(* Schneider Machine Expert - Basic project INTEGRATED_3_CONVEYOR_TM221CE24R_REV3, file version 3.0.0.0 *)
(* ProjectInformations: Name=New project *)

HARDWARE
  Cpu 0: TM221CE24R
  ModuleExtensionObject 0: TM3DI32K
  ModuleExtensionObject 1: TM3AI2H/G
  EthernetConfiguration: NetworkName=M221, IpAllocationMode=FixedAddress, IpAddress=0.0.0.0, SubnetMask=0.0.0.0
  SerialLineConfiguration: Baud=Baud19200, Parity=ParityEven, DataBits=DataBits8, StopBits=StopBits1, PhysicalMedium=PhysicalMediumRs485, TransmissionMode=TransmissionModeModbusRtu, SlaveId=1, Addressing=SlaveAddressing
  MastTask: UsePeriodScanMode=false, PeriodScan=100
  FastTask: Period=255
  CpuBehavior: StartingMode=StartAsPreviousState, AutoSaveRamOnEeprom=true, WatchdogPeriod=250

SYMBOLS  (address, symbol, comment, settings)
  %M0       AUTO_MODE  "1 Auto"
  %M1       START_HMI  "Start HMI"
  %M2       STOP_HMI  "Stop HMI"
  %M3       JOG_INFEED  "Jog infeed"
  %M4       JOG_TRANSFER  "Jog transfer"
  %M5       JOG_OUTFEED  "Jog outfeed"
  %M6       RESET_HMI  "Reset HMI"
  %M7       MAINTENANCE_ENABLE  "Izin maintenance"
  %M10      SYSTEM_RUN  "Latch produksi"
  %M11      SAFETY_OK  "Ringkasan interlock"
  %M12      OUTFEED_AUTO_CMD  "Auto command outfeed"
  %M13      TRANSFER_AUTO_CMD  "Auto command transfer"
  %M14      INFEED_AUTO_CMD  "Auto command infeed"
  %M15      INFEED_FINAL_CMD  "Final infeed"
  %M16      TRANSFER_FINAL_CMD  "Final transfer"
  %M17      OUTFEED_FINAL_CMD  "Final outfeed"
  %M20      TRANSFER_STAGE_READY  "Start delay transfer selesai"
  %M21      INFEED_STAGE_READY  "Start delay infeed selesai"
  %M22      REJECT_REQUEST  "Permintaan reject"
  %M23      REJECT_ACTIVE  "Solenoid reject aktif"
  %M24      PRODUCT_REJECTED  "Produk saat ini reject"
  %M25      EXIT_PULSE  "Pulsa exit"
  %M26      RESET_REQUEST  "Gabungan reset"
  %M30      JAM_INFEED  "Jam infeed"
  %M31      JAM_TRANSFER  "Jam transfer"
  %M32      JAM_OUTFEED  "Jam outfeed"
  %M33      REJECT_NOT_HOME  "Pusher gagal home"
  %M34      ALARM_ACTIVE  "Alarm umum"
  %M40      RESET_COUNTERS_HMI  "Reset counter produksi"
  %M41      MANUAL_INFEED_CMD  "Jog infeed tervalidasi"
  %M42      MANUAL_TRANSFER_CMD  "Jog transfer tervalidasi"
  %M43      MANUAL_OUTFEED_CMD  "Jog outfeed tervalidasi"
  %S5       SB_TB100MS  "Time base of 100 ms generated by an internal clock"
  %S6       SB_TB1S  "Time base of 1 s generated by an internal clock"
  %S13      SB_FIRSTRUN  "Indicates the first controller cycle in RUN mode"
  %MW1      WATER_RANGE_MM  "Range sensor level mm"
  %MW2      LEVEL_RAW_COPY  "Salinan raw input level"
  %MW10     MAX_HEIGHT_G1_MM  "Tinggi maksimum pintu 1 mm"
  %MW11     MAX_HEIGHT_G2_MM  "Tinggi maksimum pintu 2 mm"
  %MW12     MAX_HEIGHT_G3_MM  "Tinggi maksimum pintu 3 mm"
  %MW13     DEADBAND_PCT  "Deadband posisi persen"
  %MW20     ENC_ZERO_G1  "Nilai encoder pintu 1 saat tertutup"
  %MW21     ENC_ZERO_G2  "Nilai encoder pintu 2 saat tertutup"
  %MW22     ENC_ZERO_G3  "Nilai encoder pintu 3 saat tertutup"
  %MW23     ENC_SPAN_G1  "Span count tertutup-terbuka G1"
  %MW24     ENC_SPAN_G2  "Span count tertutup-terbuka G2"
  %MW25     ENC_SPAN_G3  "Span count tertutup-terbuka G3"
  %MW30     ENC_BINARY_G1  "Nilai biner encoder G1"
  %MW31     ENC_BINARY_G2  "Nilai biner encoder G2"
  %MW32     ENC_BINARY_G3  "Nilai biner encoder G3"
  %MW33     POS_COUNT_G1  "Count posisi terkoreksi G1"
  %MW34     POS_COUNT_G2  "Count posisi terkoreksi G2"
  %MW35     POS_COUNT_G3  "Count posisi terkoreksi G3"
  %MW50     TARGET_PCT_G1  "Target bukaan G1 0-100 persen"
  %MW51     TARGET_PCT_G2  "Target bukaan G2 0-100 persen"
  %MW52     TARGET_PCT_G3  "Target bukaan G3 0-100 persen"
  %MF60     POSITION_G1_PCT  "Posisi G1 persen"
  %MF62     POSITION_G2_PCT  "Posisi G2 persen"
  %MF64     POSITION_G3_PCT  "Posisi G3 persen"
  %MF66     POSITION_G1_MM  "Posisi G1 mm"
  %MF68     POSITION_G2_MM  "Posisi G2 mm"
  %MF70     POSITION_G3_MM  "Posisi G3 mm"
  %MF72     WATER_LEVEL_MM  "Level air mm"
  %MF74     WATER_LEVEL_PCT  "Level air persen"
  %MF76     WATER_RANGE_REAL  "Range level dalam REAL"
  %MF80     TARGET_G1_REAL  "Target G1 dalam REAL"
  %MF82     TARGET_G2_REAL  "Target G2 dalam REAL"
  %MF84     TARGET_G3_REAL  "Target G3 dalam REAL"
  %MF86     DEADBAND_REAL  "Deadband dalam REAL"
  %MF88     OPEN_THRESHOLD_G1  "Ambang buka G1"
  %MF90     CLOSE_THRESHOLD_G1  "Ambang tutup G1"
  %MF92     OPEN_THRESHOLD_G2  "Ambang buka G2"
  %MF94     CLOSE_THRESHOLD_G2  "Ambang tutup G2"
  %MF96     OPEN_THRESHOLD_G3  "Ambang buka G3"
  %MF98     CLOSE_THRESHOLD_G3  "Ambang tutup G3"
  %C0       TRANSFER_START_TICKS  "10 x 100 ms = 1 s"
  %C1       INFEED_START_TICKS  "10 x 100 ms = 1 s"
  %C2       REJECT_POSITION_TICKS  "5 x 100 ms = 0.5 s"
  %C3       REJECT_PULSE_TICKS  "7 x 100 ms = 0.7 s"
  %C4       JAM_INFEED_SECONDS  "10 x 1 s"
  %C5       JAM_TRANSFER_SECONDS  "10 x 1 s"
  %C6       JAM_OUTFEED_SECONDS  "10 x 1 s"
  %C7       REJECT_HOME_SECONDS  "3 x 1 s"
  %C8       GOOD_PRODUCT_COUNT  "Counter produk OK"
  %C9       REJECT_PRODUCT_COUNT  "Counter produk reject"
  %I0.0     START_PB  "Tombol Start NO"
  %I0.1     STOP_OK  "Kontak Stop NC; 1 sehat"
  %I0.2     ESTOP_OK  "Feedback safety relay; 1 sehat"
  %I0.3     OL_INFEED_OK  "Overload infeed; 1 sehat"
  %I0.4     OL_TRANSFER_OK  "Overload transfer; 1 sehat"
  %I0.5     OL_OUTFEED_OK  "Overload outfeed; 1 sehat"
  %I0.6     SENSOR_INFEED  "Sensor infeed"
  %I0.7     SENSOR_BUFFER1  "Sensor buffer 1"
  %I0.8     SENSOR_BUFFER2  "Sensor buffer 2"
  %I0.9     SENSOR_INSPECTION  "Sensor inspeksi"
  %I0.10    QUALITY_OK  "Hasil inspeksi OK"
  %I0.11    REJECT_HOME  "Pusher reject home"
  %I0.12    EXIT_SENSOR  "Sensor keluar"
  %I0.13    RESET_PB  "Reset alarm"
  %Q0.0     MOTOR_INFEED  "Motor conveyor infeed"
  %Q0.1     MOTOR_TRANSFER  "Motor conveyor transfer"
  %Q0.2     MOTOR_OUTFEED  "Motor conveyor outfeed"
  %Q0.3     REJECT_SOLENOID  "Solenoid reject"
  %Q0.4     BUZZER  "Buzzer fault"
  %Q0.5     LAMP_RUN  "Lampu run"
  %Q0.6     LAMP_MAINTENANCE  "Lampu maintenance"
  %Q0.7     LAMP_FAULT  "Lampu fault"
  %Q0.8       "Tidak digunakan"
  %Q0.9       "Tidak digunakan"
  %I1.0     ENC_G1_GRAY_B0  "E6CP pintu 1 Gray bit 0"
  %I1.1     ENC_G1_GRAY_B1  "E6CP pintu 1 Gray bit 1"
  %I1.2     ENC_G1_GRAY_B2  "E6CP pintu 1 Gray bit 2"
  %I1.3     ENC_G1_GRAY_B3  "E6CP pintu 1 Gray bit 3"
  %I1.4     ENC_G1_GRAY_B4  "E6CP pintu 1 Gray bit 4"
  %I1.5     ENC_G1_GRAY_B5  "E6CP pintu 1 Gray bit 5"
  %I1.6     ENC_G1_GRAY_B6  "E6CP pintu 1 Gray bit 6"
  %I1.7     ENC_G1_GRAY_B7  "E6CP pintu 1 Gray bit 7"
  %I1.8     ENC_G2_GRAY_B0  "E6CP pintu 2 Gray bit 0"
  %I1.9     ENC_G2_GRAY_B1  "E6CP pintu 2 Gray bit 1"
  %I1.10    ENC_G2_GRAY_B2  "E6CP pintu 2 Gray bit 2"
  %I1.11    ENC_G2_GRAY_B3  "E6CP pintu 2 Gray bit 3"
  %I1.12    ENC_G2_GRAY_B4  "E6CP pintu 2 Gray bit 4"
  %I1.13    ENC_G2_GRAY_B5  "E6CP pintu 2 Gray bit 5"
  %I1.14    ENC_G2_GRAY_B6  "E6CP pintu 2 Gray bit 6"
  %I1.15    ENC_G2_GRAY_B7  "E6CP pintu 2 Gray bit 7"
  %I1.16    ENC_G3_GRAY_B0  "E6CP pintu 3 Gray bit 0"
  %I1.17    ENC_G3_GRAY_B1  "E6CP pintu 3 Gray bit 1"
  %I1.18    ENC_G3_GRAY_B2  "E6CP pintu 3 Gray bit 2"
  %I1.19    ENC_G3_GRAY_B3  "E6CP pintu 3 Gray bit 3"
  %I1.20    ENC_G3_GRAY_B4  "E6CP pintu 3 Gray bit 4"
  %I1.21    ENC_G3_GRAY_B5  "E6CP pintu 3 Gray bit 5"
  %I1.22    ENC_G3_GRAY_B6  "E6CP pintu 3 Gray bit 6"
  %I1.23    ENC_G3_GRAY_B7  "E6CP pintu 3 Gray bit 7"
  %I1.24    MODE_AUTO  "Selector 1=AUTO 0=MANUAL"
  %I1.25    MAN_OPEN_G1  "PB manual buka pintu 1"
  %I1.26    MAN_CLOSE_G1  "PB manual tutup pintu 1"
  %I1.27    MAN_OPEN_G2  "PB manual buka pintu 2"
  %I1.28    MAN_CLOSE_G2  "PB manual tutup pintu 2"
  %I1.29    MAN_OPEN_G3  "PB manual buka pintu 3"
  %I1.30    MAN_CLOSE_G3  "PB manual tutup pintu 3"
  %I1.31    RESET_FAULT  "PB reset fault"
  %IW2.0    LEVEL_RAW  "Sensor level 4-20 mA raw 4000-20000"  [Type=Type_4_20mA, Scope=Scope_Customized, Minimum=4000, Maximum=20000]

POU INTEGRATED_3_CONVEYOR_IL
  (* SectionNumber=1 *)

// Rung 0: N01_SAFETY
// Stop, E-Stop, dan tiga overload.
  LD %I0.1                (* STOP_OK *)
  AND %I0.2               (* ESTOP_OK *)
  AND %I0.3               (* OL_INFEED_OK *)
  AND %I0.4               (* OL_TRANSFER_OK *)
  AND %I0.5               (* OL_OUTFEED_OK *)
  ANDN %M2                (* STOP_HMI *)
  ST %M11                 (* SAFETY_OK *)
  // as ST:
  //   SAFETY_OK := STOP_OK AND ESTOP_OK AND OL_INFEED_OK AND OL_TRANSFER_OK AND OL_OUTFEED_OK AND NOT STOP_HMI;

// Rung 1: N02_SYSTEM_RUN
// Latch produksi Auto.
  LD %I0.0                (* START_PB *)
  OR %M1                  (* START_HMI *)
  OR %M10                 (* SYSTEM_RUN *)
  AND %M0                 (* AUTO_MODE *)
  AND %M11                (* SAFETY_OK *)
  ST %M10                 (* SYSTEM_RUN *)
  // as ST:
  //   SYSTEM_RUN := (START_PB OR START_HMI OR SYSTEM_RUN) AND AUTO_MODE AND SAFETY_OK;

// Rung 2: N03_RESET
// Gabungan reset.
  LD %I0.13               (* RESET_PB *)
  OR %M6                  (* RESET_HMI *)
  ST %M26                 (* RESET_REQUEST *)
  // as ST:
  //   RESET_REQUEST := RESET_PB OR RESET_HMI;

// Rung 3: N04_OUTFEED_BASE
// Hilir start lebih dahulu.
  LD %M10                 (* SYSTEM_RUN *)
  ANDN %M34               (* ALARM_ACTIVE *)
  ST %M12                 (* OUTFEED_AUTO_CMD *)
  // as ST:
  //   OUTFEED_AUTO_CMD := SYSTEM_RUN AND NOT ALARM_ACTIVE;

// Rung 4: N05_PRESET_C0
// Preset transfer start.
  LD %S13                 (* SB_FIRSTRUN *)
  [ %C0.P := 10 ]         (* TRANSFER_START_TICKS *)
  // as ST:
  //   IF SB_FIRSTRUN THEN TRANSFER_START_TICKS.P := 10; END_IF;

// Rung 5: N05_PRESET_C1
// Preset infeed start.
  LD %S13                 (* SB_FIRSTRUN *)
  [ %C1.P := 10 ]         (* INFEED_START_TICKS *)
  // as ST:
  //   IF SB_FIRSTRUN THEN INFEED_START_TICKS.P := 10; END_IF;

// Rung 6: N05_PRESET_C2
// Preset posisi reject.
  LD %S13                 (* SB_FIRSTRUN *)
  [ %C2.P := 5 ]          (* REJECT_POSITION_TICKS *)
  // as ST:
  //   IF SB_FIRSTRUN THEN REJECT_POSITION_TICKS.P := 5; END_IF;

// Rung 7: N05_PRESET_C3
// Preset pulsa reject.
  LD %S13                 (* SB_FIRSTRUN *)
  [ %C3.P := 7 ]          (* REJECT_PULSE_TICKS *)
  // as ST:
  //   IF SB_FIRSTRUN THEN REJECT_PULSE_TICKS.P := 7; END_IF;

// Rung 8: N05_PRESET_C4
// Preset jam infeed.
  LD %S13                 (* SB_FIRSTRUN *)
  [ %C4.P := 10 ]         (* JAM_INFEED_SECONDS *)
  // as ST:
  //   IF SB_FIRSTRUN THEN JAM_INFEED_SECONDS.P := 10; END_IF;

// Rung 9: N05_PRESET_C5
// Preset jam transfer.
  LD %S13                 (* SB_FIRSTRUN *)
  [ %C5.P := 10 ]         (* JAM_TRANSFER_SECONDS *)
  // as ST:
  //   IF SB_FIRSTRUN THEN JAM_TRANSFER_SECONDS.P := 10; END_IF;

// Rung 10: N05_PRESET_C6
// Preset jam outfeed.
  LD %S13                 (* SB_FIRSTRUN *)
  [ %C6.P := 10 ]         (* JAM_OUTFEED_SECONDS *)
  // as ST:
  //   IF SB_FIRSTRUN THEN JAM_OUTFEED_SECONDS.P := 10; END_IF;

// Rung 11: N05_PRESET_C7
// Preset pusher home.
  LD %S13                 (* SB_FIRSTRUN *)
  [ %C7.P := 3 ]          (* REJECT_HOME_SECONDS *)
  // as ST:
  //   IF SB_FIRSTRUN THEN REJECT_HOME_SECONDS.P := 3; END_IF;

// Rung 12: N06_TRANSFER_DELAY
// Delay 1 detik.
  BLK %C0                 (* TRANSFER_START_TICKS *)
  LD %S5                  (* SB_TB100MS *)
  AND %M12                (* OUTFEED_AUTO_CMD *)
  CU
  LDN %M12                (* OUTFEED_AUTO_CMD *)
  R
  END_BLK
  // as ST:
  //   TRANSFER_START_TICKS(CU := SB_TB100MS AND OUTFEED_AUTO_CMD, R := NOT OUTFEED_AUTO_CMD);

// Rung 13: N07_TRANSFER_READY
// Transfer siap.
  LD %C0.D                (* TRANSFER_START_TICKS *)
  ST %M20                 (* TRANSFER_STAGE_READY *)
  // as ST:
  //   TRANSFER_STAGE_READY := TRANSFER_START_TICKS.D;

// Rung 14: N09_INFEED_DELAY
// Delay 1 detik setelah transfer.
  BLK %C1                 (* INFEED_START_TICKS *)
  LD %S5                  (* SB_TB100MS *)
  AND %M20                (* TRANSFER_STAGE_READY *)
  CU
  LDN %M20                (* TRANSFER_STAGE_READY *)
  R
  END_BLK
  // as ST:
  //   INFEED_START_TICKS(CU := SB_TB100MS AND TRANSFER_STAGE_READY, R := NOT TRANSFER_STAGE_READY);

// Rung 15: N10_INFEED_READY
// Infeed siap.
  LD %C1.D                (* INFEED_START_TICKS *)
  ST %M21                 (* INFEED_STAGE_READY *)
  // as ST:
  //   INFEED_STAGE_READY := INFEED_START_TICKS.D;

// Rung 16: N11_INFEED_AUTO
// Kontrol buffer 1 Auto.
  LD %M21                 (* INFEED_STAGE_READY *)
  ANDN %I0.7              (* SENSOR_BUFFER1 *)
  ANDN %M34               (* ALARM_ACTIVE *)
  ST %M14                 (* INFEED_AUTO_CMD *)
  // as ST:
  //   INFEED_AUTO_CMD := INFEED_STAGE_READY AND NOT SENSOR_BUFFER1 AND NOT ALARM_ACTIVE;

// Rung 17: N12_TRANSFER_AUTO
// Kontrol buffer 2 Auto.
  LD %M20                 (* TRANSFER_STAGE_READY *)
  ANDN %I0.8              (* SENSOR_BUFFER2 *)
  ANDN %M34               (* ALARM_ACTIVE *)
  ST %M13                 (* TRANSFER_AUTO_CMD *)
  // as ST:
  //   TRANSFER_AUTO_CMD := TRANSFER_STAGE_READY AND NOT SENSOR_BUFFER2 AND NOT ALARM_ACTIVE;

// Rung 18: N13_REJECT_CAPTURE
// Latch produk NG.
  LDR %I0.9               (* SENSOR_INSPECTION *)
  ANDN %I0.10             (* QUALITY_OK *)
  AND %M10                (* SYSTEM_RUN *)
  S %M22                  (* REJECT_REQUEST *)
  S %M24                  (* PRODUCT_REJECTED *)
  // as ST:
  //   IF RISING(SENSOR_INSPECTION) AND NOT QUALITY_OK AND SYSTEM_RUN THEN REJECT_REQUEST := TRUE; END_IF;
  //   IF RISING(SENSOR_INSPECTION) AND NOT QUALITY_OK AND SYSTEM_RUN THEN PRODUCT_REJECTED := TRUE; END_IF;

// Rung 19: N14_REJECT_POSITION
// Delay produk ke pusher.
  BLK %C2                 (* REJECT_POSITION_TICKS *)
  LD %S5                  (* SB_TB100MS *)
  AND %M22                (* REJECT_REQUEST *)
  AND %I0.11              (* REJECT_HOME *)
  CU
  LDN %M22                (* REJECT_REQUEST *)
  ORN %I0.11              (* REJECT_HOME *)
  R
  END_BLK
  // as ST:
  //   REJECT_POSITION_TICKS(CU := SB_TB100MS AND REJECT_REQUEST AND REJECT_HOME, R := NOT REJECT_REQUEST OR NOT REJECT_HOME);

// Rung 20: N15_REJECT_START
// Mulai aktuator.
  LD %C2.D                (* REJECT_POSITION_TICKS *)
  S %M23                  (* REJECT_ACTIVE *)
  // as ST:
  //   IF REJECT_POSITION_TICKS.D THEN REJECT_ACTIVE := TRUE; END_IF;

// Rung 21: N17_REJECT_PULSE
// Durasi aktuator.
  BLK %C3                 (* REJECT_PULSE_TICKS *)
  LD %S5                  (* SB_TB100MS *)
  AND %M23                (* REJECT_ACTIVE *)
  CU
  LDN %M23                (* REJECT_ACTIVE *)
  R
  END_BLK
  // as ST:
  //   REJECT_PULSE_TICKS(CU := SB_TB100MS AND REJECT_ACTIVE, R := NOT REJECT_ACTIVE);

// Rung 22: N18_REJECT_DONE
// Akhiri reject request.
  LD %C3.D                (* REJECT_PULSE_TICKS *)
  R %M23                  (* REJECT_ACTIVE *)
  R %M22                  (* REJECT_REQUEST *)
  // as ST:
  //   IF REJECT_PULSE_TICKS.D THEN REJECT_ACTIVE := FALSE; END_IF;
  //   IF REJECT_PULSE_TICKS.D THEN REJECT_REQUEST := FALSE; END_IF;

// Rung 23: N20_JAM_INFEED_COUNTER
// Monitor buffer 1.
  BLK %C4                 (* JAM_INFEED_SECONDS *)
  LD %S6                  (* SB_TB1S *)
  AND %M14                (* INFEED_AUTO_CMD *)
  AND %I0.7               (* SENSOR_BUFFER1 *)
  CU
  LDN %M14                (* INFEED_AUTO_CMD *)
  ORN %I0.7               (* SENSOR_BUFFER1 *)
  R
  END_BLK
  // as ST:
  //   JAM_INFEED_SECONDS(CU := SB_TB1S AND INFEED_AUTO_CMD AND SENSOR_BUFFER1, R := NOT INFEED_AUTO_CMD OR NOT SENSOR_BUFFER1);

// Rung 24: N22_JAM_TRANSFER_COUNTER
// Monitor buffer 2.
  BLK %C5                 (* JAM_TRANSFER_SECONDS *)
  LD %S6                  (* SB_TB1S *)
  AND %M13                (* TRANSFER_AUTO_CMD *)
  AND %I0.8               (* SENSOR_BUFFER2 *)
  CU
  LDN %M13                (* TRANSFER_AUTO_CMD *)
  ORN %I0.8               (* SENSOR_BUFFER2 *)
  R
  END_BLK
  // as ST:
  //   JAM_TRANSFER_SECONDS(CU := SB_TB1S AND TRANSFER_AUTO_CMD AND SENSOR_BUFFER2, R := NOT TRANSFER_AUTO_CMD OR NOT SENSOR_BUFFER2);

// Rung 25: N24_JAM_OUTFEED_COUNTER
// Monitor exit.
  BLK %C6                 (* JAM_OUTFEED_SECONDS *)
  LD %S6                  (* SB_TB1S *)
  AND %M12                (* OUTFEED_AUTO_CMD *)
  AND %I0.12              (* EXIT_SENSOR *)
  CU
  LDN %M12                (* OUTFEED_AUTO_CMD *)
  ORN %I0.12              (* EXIT_SENSOR *)
  R
  END_BLK
  // as ST:
  //   JAM_OUTFEED_SECONDS(CU := SB_TB1S AND OUTFEED_AUTO_CMD AND EXIT_SENSOR, R := NOT OUTFEED_AUTO_CMD OR NOT EXIT_SENSOR);

// Rung 26: N26_HOME_TIMEOUT_COUNTER
// Pusher harus kembali home.
  BLK %C7                 (* REJECT_HOME_SECONDS *)
  LD %S6                  (* SB_TB1S *)
  AND %M24                (* PRODUCT_REJECTED *)
  ANDN %M23               (* REJECT_ACTIVE *)
  ANDN %I0.11             (* REJECT_HOME *)
  CU
  LDN %M24                (* PRODUCT_REJECTED *)
  OR %I0.11               (* REJECT_HOME *)
  R
  END_BLK
  // as ST:
  //   REJECT_HOME_SECONDS(CU := SB_TB1S AND PRODUCT_REJECTED AND NOT REJECT_ACTIVE AND NOT REJECT_HOME, R := NOT PRODUCT_REJECTED OR REJECT_HOME);

// Rung 27: N27_LATCH_JAM_INFEED
// Latch jam infeed.
  LD %C4.D                (* JAM_INFEED_SECONDS *)
  S %M30                  (* JAM_INFEED *)
  // as ST:
  //   IF JAM_INFEED_SECONDS.D THEN JAM_INFEED := TRUE; END_IF;

// Rung 28: N28_LATCH_JAM_TRANSFER
// Latch jam transfer.
  LD %C5.D                (* JAM_TRANSFER_SECONDS *)
  S %M31                  (* JAM_TRANSFER *)
  // as ST:
  //   IF JAM_TRANSFER_SECONDS.D THEN JAM_TRANSFER := TRUE; END_IF;

// Rung 29: N29_LATCH_JAM_OUTFEED
// Latch jam outfeed.
  LD %C6.D                (* JAM_OUTFEED_SECONDS *)
  S %M32                  (* JAM_OUTFEED *)
  // as ST:
  //   IF JAM_OUTFEED_SECONDS.D THEN JAM_OUTFEED := TRUE; END_IF;

// Rung 30: N30_LATCH_HOME_FAULT
// Latch pusher tidak home.
  LD %C7.D                (* REJECT_HOME_SECONDS *)
  S %M33                  (* REJECT_NOT_HOME *)
  // as ST:
  //   IF REJECT_HOME_SECONDS.D THEN REJECT_NOT_HOME := TRUE; END_IF;

// Rung 31: N31_RESET_JAM_INFEED
// Reset jam infeed saat sensor pulih.
  LD %M26                 (* RESET_REQUEST *)
  ANDN %I0.7              (* SENSOR_BUFFER1 *)
  R %M30                  (* JAM_INFEED *)
  // as ST:
  //   IF RESET_REQUEST AND NOT SENSOR_BUFFER1 THEN JAM_INFEED := FALSE; END_IF;

// Rung 32: N32_RESET_JAM_TRANSFER
// Reset jam transfer saat sensor pulih.
  LD %M26                 (* RESET_REQUEST *)
  ANDN %I0.8              (* SENSOR_BUFFER2 *)
  R %M31                  (* JAM_TRANSFER *)
  // as ST:
  //   IF RESET_REQUEST AND NOT SENSOR_BUFFER2 THEN JAM_TRANSFER := FALSE; END_IF;

// Rung 33: N33_RESET_JAM_OUTFEED
// Reset jam outfeed saat sensor pulih.
  LD %M26                 (* RESET_REQUEST *)
  ANDN %I0.12             (* EXIT_SENSOR *)
  R %M32                  (* JAM_OUTFEED *)
  // as ST:
  //   IF RESET_REQUEST AND NOT EXIT_SENSOR THEN JAM_OUTFEED := FALSE; END_IF;

// Rung 34: N34_RESET_HOME_FAULT
// Reset fault saat pusher home.
  LD %M26                 (* RESET_REQUEST *)
  AND %I0.11              (* REJECT_HOME *)
  R %M33                  (* REJECT_NOT_HOME *)
  // as ST:
  //   IF RESET_REQUEST AND REJECT_HOME THEN REJECT_NOT_HOME := FALSE; END_IF;

// Rung 35: N35_ALARM
// Ringkasan alarm.
  LD %M30                 (* JAM_INFEED *)
  OR %M31                 (* JAM_TRANSFER *)
  OR %M32                 (* JAM_OUTFEED *)
  OR %M33                 (* REJECT_NOT_HOME *)
  ORN %I0.2               (* ESTOP_OK *)
  ORN %I0.3               (* OL_INFEED_OK *)
  ORN %I0.4               (* OL_TRANSFER_OK *)
  ORN %I0.5               (* OL_OUTFEED_OK *)
  ST %M34                 (* ALARM_ACTIVE *)
  // as ST:
  //   ALARM_ACTIVE := JAM_INFEED OR JAM_TRANSFER OR JAM_OUTFEED OR REJECT_NOT_HOME OR NOT ESTOP_OK OR NOT OL_INFEED_OK OR NOT OL_TRANSFER_OK OR NOT OL_OUTFEED_OK;

// Rung 36: N36_MANUAL_INFEED
// Jog maintenance infeed.
  LD %M3                  (* JOG_INFEED *)
  ANDN %M0                (* AUTO_MODE *)
  AND %M7                 (* MAINTENANCE_ENABLE *)
  ST %M41                 (* MANUAL_INFEED_CMD *)
  // as ST:
  //   MANUAL_INFEED_CMD := JOG_INFEED AND NOT AUTO_MODE AND MAINTENANCE_ENABLE;

// Rung 37: N37_MANUAL_TRANSFER
// Jog maintenance transfer.
  LD %M4                  (* JOG_TRANSFER *)
  ANDN %M0                (* AUTO_MODE *)
  AND %M7                 (* MAINTENANCE_ENABLE *)
  ST %M42                 (* MANUAL_TRANSFER_CMD *)
  // as ST:
  //   MANUAL_TRANSFER_CMD := JOG_TRANSFER AND NOT AUTO_MODE AND MAINTENANCE_ENABLE;

// Rung 38: N38_MANUAL_OUTFEED
// Jog maintenance outfeed.
  LD %M5                  (* JOG_OUTFEED *)
  ANDN %M0                (* AUTO_MODE *)
  AND %M7                 (* MAINTENANCE_ENABLE *)
  ST %M43                 (* MANUAL_OUTFEED_CMD *)
  // as ST:
  //   MANUAL_OUTFEED_CMD := JOG_OUTFEED AND NOT AUTO_MODE AND MAINTENANCE_ENABLE;

// Rung 39: N39_FINAL_INFEED
// Auto atau jog infeed.
  LD %M14                 (* INFEED_AUTO_CMD *)
  OR %M41                 (* MANUAL_INFEED_CMD *)
  AND %M11                (* SAFETY_OK *)
  ANDN %M34               (* ALARM_ACTIVE *)
  ST %M15                 (* INFEED_FINAL_CMD *)
  // as ST:
  //   INFEED_FINAL_CMD := (INFEED_AUTO_CMD OR MANUAL_INFEED_CMD) AND SAFETY_OK AND NOT ALARM_ACTIVE;

// Rung 40: N40_FINAL_TRANSFER
// Auto atau jog transfer.
  LD %M13                 (* TRANSFER_AUTO_CMD *)
  OR %M42                 (* MANUAL_TRANSFER_CMD *)
  AND %M11                (* SAFETY_OK *)
  ANDN %M34               (* ALARM_ACTIVE *)
  ST %M16                 (* TRANSFER_FINAL_CMD *)
  // as ST:
  //   TRANSFER_FINAL_CMD := (TRANSFER_AUTO_CMD OR MANUAL_TRANSFER_CMD) AND SAFETY_OK AND NOT ALARM_ACTIVE;

// Rung 41: N41_FINAL_OUTFEED
// Auto atau jog outfeed.
  LD %M12                 (* OUTFEED_AUTO_CMD *)
  OR %M43                 (* MANUAL_OUTFEED_CMD *)
  AND %M11                (* SAFETY_OK *)
  ANDN %M34               (* ALARM_ACTIVE *)
  ST %M17                 (* OUTFEED_FINAL_CMD *)
  // as ST:
  //   OUTFEED_FINAL_CMD := (OUTFEED_AUTO_CMD OR MANUAL_OUTFEED_CMD) AND SAFETY_OK AND NOT ALARM_ACTIVE;

// Rung 42: N42_OUTPUT_INFEED
// Output motor infeed.
  LD %M15                 (* INFEED_FINAL_CMD *)
  ST %Q0.0                (* MOTOR_INFEED *)
  // as ST:
  //   MOTOR_INFEED := INFEED_FINAL_CMD;

// Rung 43: N43_OUTPUT_TRANSFER
// Output motor transfer.
  LD %M16                 (* TRANSFER_FINAL_CMD *)
  ST %Q0.1                (* MOTOR_TRANSFER *)
  // as ST:
  //   MOTOR_TRANSFER := TRANSFER_FINAL_CMD;

// Rung 44: N44_OUTPUT_OUTFEED
// Output motor outfeed.
  LD %M17                 (* OUTFEED_FINAL_CMD *)
  ST %Q0.2                (* MOTOR_OUTFEED *)
  // as ST:
  //   MOTOR_OUTFEED := OUTFEED_FINAL_CMD;

// Rung 45: N45_OUTPUT_REJECT
// Output solenoid reject.
  LD %M23                 (* REJECT_ACTIVE *)
  AND %M11                (* SAFETY_OK *)
  ANDN %M34               (* ALARM_ACTIVE *)
  ST %Q0.3                (* REJECT_SOLENOID *)
  // as ST:
  //   REJECT_SOLENOID := REJECT_ACTIVE AND SAFETY_OK AND NOT ALARM_ACTIVE;

// Rung 46: N46_EXIT_PULSE
// Pulsa produk keluar.
  LDR %I0.12              (* EXIT_SENSOR *)
  ST %M25                 (* EXIT_PULSE *)
  // as ST:
  //   EXIT_PULSE := RISING(EXIT_SENSOR);

// Rung 47: N47_COUNT_GOOD
// Counter produk OK.
  BLK %C8                 (* GOOD_PRODUCT_COUNT *)
  LD %M25                 (* EXIT_PULSE *)
  ANDN %M24               (* PRODUCT_REJECTED *)
  CU
  LD %M40                 (* RESET_COUNTERS_HMI *)
  R
  END_BLK
  // as ST:
  //   GOOD_PRODUCT_COUNT(CU := EXIT_PULSE AND NOT PRODUCT_REJECTED, R := RESET_COUNTERS_HMI);

// Rung 48: N48_COUNT_REJECT
// Counter produk reject.
  BLK %C9                 (* REJECT_PRODUCT_COUNT *)
  LD %M25                 (* EXIT_PULSE *)
  AND %M24                (* PRODUCT_REJECTED *)
  CU
  LD %M40                 (* RESET_COUNTERS_HMI *)
  R
  END_BLK
  // as ST:
  //   REJECT_PRODUCT_COUNT(CU := EXIT_PULSE AND PRODUCT_REJECTED, R := RESET_COUNTERS_HMI);

// Rung 49: N49_CLEAR_PRODUCT
// Selesai tracking produk.
  LD %M25                 (* EXIT_PULSE *)
  R %M24                  (* PRODUCT_REJECTED *)
  // as ST:
  //   IF EXIT_PULSE THEN PRODUCT_REJECTED := FALSE; END_IF;

// Rung 50: N50_LAMP_RUN
// Lampu run.
  LD %M10                 (* SYSTEM_RUN *)
  ANDN %M34               (* ALARM_ACTIVE *)
  ST %Q0.5                (* LAMP_RUN *)
  // as ST:
  //   LAMP_RUN := SYSTEM_RUN AND NOT ALARM_ACTIVE;

// Rung 51: N51_LAMP_MAINT
// Lampu maintenance.
  LDN %M0                 (* AUTO_MODE *)
  AND %M7                 (* MAINTENANCE_ENABLE *)
  ST %Q0.6                (* LAMP_MAINTENANCE *)
  // as ST:
  //   LAMP_MAINTENANCE := NOT AUTO_MODE AND MAINTENANCE_ENABLE;

// Rung 52: N52_FAULT_OUTPUTS
// Lampu fault dan buzzer.
  LD %M34                 (* ALARM_ACTIVE *)
  ST %Q0.7                (* LAMP_FAULT *)
  ST %Q0.4                (* BUZZER *)
  // as ST:
  //   LAMP_FAULT := ALARM_ACTIVE;
  //   BUZZER := ALARM_ACTIVE;
